(* PLC project manufacturing, Dassault Systèmes ControlBuild 2024x Refresh1 *)
(* stored: creationDateTime 2024-04-12T14:05:59-01:00 *)

FUNCTION_BLOCK faults
  VAR_INPUT
    fault3 : BOOL := false;
    fault2 : BOOL := false;
    fault1 : BOOL := false;
  END_VAR
  VAR_OUTPUT
    generalFault : BOOL := false;
  END_VAR

(* LD diagram, written out as Structured Text *)
1:
generalFault := fault3 OR fault1 OR fault2;
END_FUNCTION_BLOCK

PROGRAM copie_batch.manufacturing
  VAR_INPUT
    cycleInProgress : BOOL := false;
    acknowledgePB : BOOL := false;
    flourWeighingRequest : BOOL := false;
    syrupWeighingRequest : BOOL := false;
    kneadingRequest : BOOL := false;
  END_VAR
  VAR_INPUT
    autoMode : BOOL := false;
    manualMode : BOOL := false;
  END_VAR
  VAR_INPUT
    flourWeight : DINT := 0;
  END_VAR
  VAR_INPUT
    syrup1Weight : DINT := 0;
    syrup2Weight : DINT := 0;
    syrup3Weight : DINT := 0;
  END_VAR
  VAR_OUTPUT
    generalFault : BOOL := false;
    kneadingOK : BOOL := false;
    flourWeighingOk : BOOL := false;
    syrupWeighingOk : BOOL := false;
  END_VAR

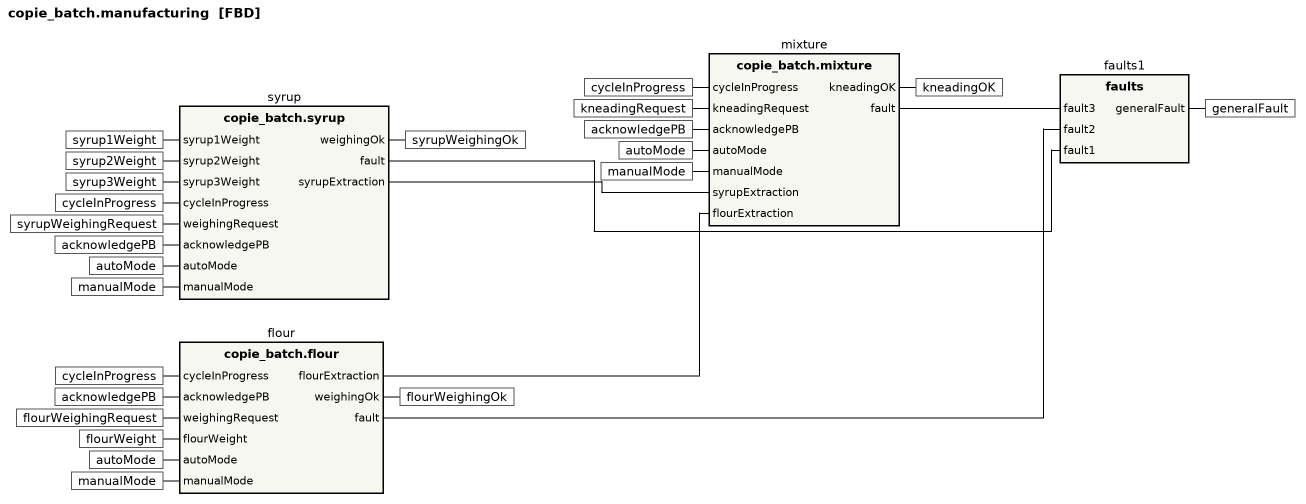
(* FBD diagram, written out as Structured Text *)
flour(cycleInProgress := cycleInProgress, acknowledgePB := acknowledgePB, weighingRequest := flourWeighingRequest, flourWeight := flourWeight, autoMode := autoMode, manualMode := manualMode);
flourWeighingOk := flour.weighingOk;
syrup(syrup1Weight := syrup1Weight, syrup2Weight := syrup2Weight, syrup3Weight := syrup3Weight, cycleInProgress := cycleInProgress, weighingRequest := syrupWeighingRequest, acknowledgePB := acknowledgePB, autoMode := autoMode, manualMode := manualMode);
mixture(cycleInProgress := cycleInProgress, kneadingRequest := kneadingRequest, acknowledgePB := acknowledgePB, autoMode := autoMode, manualMode := manualMode, syrupExtraction := syrup.syrupExtraction, flourExtraction := flour.flourExtraction);
kneadingOK := mixture.kneadingOK;
faults1(fault3 := mixture.fault, fault2 := flour.fault, fault1 := syrup.fault);
generalFault := faults1.generalFault;
syrupWeighingOk := syrup.weighingOk;
END_PROGRAM
